// TIA Portal V20 export
DATA_BLOCK "SBK09"   // DB326
// stored: MemoryReserve 100
   VAR
      "SAFETY DOOR LOCK4.INPUT" : Bool := TRUE;
      "SAFETY DOOR LOCK5.INPUT" : Bool := TRUE;
      "SAFETY DOOR LOCK6.INPUT" : Bool := TRUE;
      SPARE : Bool := FALSE;
      "SAFETY DOOR LOCK4.INPUT_1" : Bool := FALSE;
      "SAFETY DOOR LOCK5.INPUT_1" : Bool := FALSE;
      "SAFETY DOOR LOCK6.INPUT_1" : Bool := FALSE;
      SPARE_1 : Bool := FALSE;
      "SAFETY DOOR LOCK4.OUTPUT" : Bool := FALSE;
      "SAFETY DOOR LOCK5.OUTPUT" : Bool := FALSE;
      "SAFETY DOOR LOCK6.OUTPUT" : Bool := FALSE;
   END_VAR
BEGIN
END_DATA_BLOCK
